FUNCTION_BLOCK FB_LamparaMemorizada_SFC_2
// La lampara se enciende al accionar el pulsador de conexion
// La lampara se apaga al accionar el pulsador de desconexion
VAR
    Lampara AT %Q*: BOOL;
    PulsadorConexion AT %I*: BOOL;
    PulsadorDesconexion AT %I*: BOOL;
END_VAR

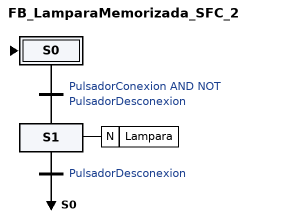
INITIAL_STEP S0:
END_STEP
TRANSITION FROM S0 TO S1
    := PulsadorConexion AND NOT PulsadorDesconexion;
END_TRANSITION
STEP S1:
    Lampara(N);
END_STEP
TRANSITION FROM S1 TO S0
    := PulsadorDesconexion;
END_TRANSITION

END_FUNCTION_BLOCK

(* stored: Version 1.1.0.1, ProductVersion 3.1.4024.15
   POU FB_LamparaMemorizada_SFC_2: Id {5dc7e891-deec-46d2-bf0e-dc9d2fcd12ee}, SpecialFunc None *)
